(* IEC 61131-3 sources: beckhoffAutomationInterface/ST/Shark/Lib/Hardware/SMC, 2 files *)

(* ---- FB_SMCAdapter.st ---- *)
(* Adapter to treat a bit in an SMC Output Block as a standard I_DigitalOutput. *)
FUNCTION_BLOCK FB_SMCAdapter IMPLEMENTS I_DigitalOutput
VAR
    _refBlock     : REFERENCE TO FB_SMCOutputBlock;
    _nIndex       : USINT;
    _bSafeState   : BOOL := FALSE;   // Applied by SetSafeState() — configured at Init time
    _bInitialized : BOOL := FALSE;
END_VAR

METHOD PUBLIC Init : BOOL
VAR_INPUT
    refBlock   : REFERENCE TO FB_SMCOutputBlock;
    nIndex     : USINT;
    bSafeState : BOOL := FALSE;   // Output state applied when SetSafeState() is called
END_VAR
    IF NOT __ISVALIDREF(refBlock) THEN
        Init := FALSE;
        RETURN;
    END_IF

    _refBlock REF= refBlock;
    _nIndex := nIndex;
    _bSafeState := bSafeState;
    _bInitialized := TRUE;
    Init := TRUE;
END_METHOD

METHOD PUBLIC SetOutput
VAR_INPUT
    bValue : BOOL;
END_VAR
    IF _bInitialized THEN
        _refBlock.SetOutput(_nIndex, bValue);
    END_IF
END_METHOD

METHOD PUBLIC GetOutput : BOOL
    IF _bInitialized THEN
        GetOutput := _refBlock.GetOutput(_nIndex);
    ELSE
        GetOutput := FALSE;
    END_IF
END_METHOD

METHOD PUBLIC SetSafeState
    IF _bInitialized THEN
        _refBlock.SetOutput(_nIndex, _bSafeState);
    END_IF
END_METHOD

END_FUNCTION_BLOCK

(* ---- FB_SMCOutputBlock.st ---- *)
(* SMC EtherCAT output block - manages 32 digital outputs via 4 bytes. *)
FUNCTION_BLOCK FB_SMCOutputBlock
VAR_IN_OUT
    aOutputBytes : ARRAY[0..3] OF BYTE;
END_VAR
VAR_OUTPUT
    bError     : BOOL;
    eErrorId   : E_ErrorId;
END_VAR
VAR
    _pOutputBytes : POINTER TO ARRAY[0..3] OF BYTE;
END_VAR
VAR CONSTANT
    MAX_OUTPUTS : USINT := 32;
END_VAR

    // Capture the address of the IN_OUT variable during FB execution
    _pOutputBytes := ADR(aOutputBytes);

METHOD PUBLIC SetOutput : BOOL
VAR_INPUT
    nIndex : USINT;
    bState : BOOL;
END_VAR
VAR
    nByteIdx : USINT;
    nBitIdx  : USINT;
END_VAR
    IF nIndex >= MAX_OUTPUTS THEN
        bError := TRUE;
        eErrorId := E_ErrorId.ERR_VALVE_INVALID_INDEX;
        SetOutput := FALSE;
        RETURN;
    END_IF

    // Check if pointer is valid (FB must be executed at least once)
    IF _pOutputBytes = 0 THEN
        bError := TRUE;
        eErrorId := E_ErrorId.ERR_GEN_NULL_POINTER;
        SetOutput := FALSE;
        RETURN;
    END_IF

    nByteIdx := nIndex / 8;
    nBitIdx := nIndex MOD 8;

    IF bState THEN
        _pOutputBytes^[nByteIdx] := _pOutputBytes^[nByteIdx] OR SHL(USINT_TO_BYTE(1), nBitIdx);
    ELSE
        _pOutputBytes^[nByteIdx] := _pOutputBytes^[nByteIdx] AND NOT SHL(USINT_TO_BYTE(1), nBitIdx);
    END_IF

    SetOutput := TRUE;
END_METHOD

METHOD PUBLIC GetOutput : BOOL
VAR_INPUT
    nIndex : USINT;
END_VAR
VAR
    nByteIdx : USINT;
    nBitIdx  : USINT;
END_VAR
    IF nIndex >= MAX_OUTPUTS THEN
        bError := TRUE;
        eErrorId := E_ErrorId.ERR_VALVE_INVALID_INDEX;
        GetOutput := FALSE;
        RETURN;
    END_IF

    IF _pOutputBytes = 0 THEN
        bError := TRUE;
        eErrorId := E_ErrorId.ERR_GEN_NULL_POINTER;
        GetOutput := FALSE;
        RETURN;
    END_IF

    nByteIdx := nIndex / 8;
    nBitIdx := nIndex MOD 8;

    GetOutput := (_pOutputBytes^[nByteIdx] AND SHL(USINT_TO_BYTE(1), nBitIdx)) <> 0;
END_METHOD

METHOD PUBLIC ClearAll
    IF _pOutputBytes = 0 THEN
        RETURN;
    END_IF

    _pOutputBytes^[0] := 0;
    _pOutputBytes^[1] := 0;
    _pOutputBytes^[2] := 0;
    _pOutputBytes^[3] := 0;
END_METHOD

METHOD PUBLIC ClearError
    bError := FALSE;
    eErrorId := E_ErrorId.NO_ERROR;
END_METHOD

END_FUNCTION_BLOCK
